PROGRAM P_SqlSelect
VAR
	
	fbSq : FB_EasySql;
	sSql : STRING(1000);
	
	iGE : INT:=1; //Select value
	
	astData : ARRAY[0..9] OF ST_SelectStruct; //Data array for recieved data
	
	bRead : BOOL; //Execute command
	bDone : BOOL; //Command done
	bError : BOOL; //Command error
	sError : STRING(255);
	
	udiNoOfRecords : UDINT; //Numbers of returned recoreds
	
END_VAR

//Select data from database
sSql := 'SELECT id,username,password FROM tpr_db.user where id >=¤1¤';

F_Replace(pString:= ADR(sSql), cbStringLen:= SIZEOF(sSql), sSearch:= '¤1¤', sReplace:= TO_STRING(iGE)); //Replace placeholder

fbSq(
	bExecute:= bRead, 
	wDBID:= 1, 
	pSql:= ADR(sSql), 
	cbSql:= SIZEOF(sSql), 
	pData:= ADR(astData), 
	cbData:= SIZEOF(astData), 
	udiMaxOfRecord:= 3, //Max number of recieved records
	udiNoOfRecords=> udiNoOfRecords, 
	bDone=> bDone, 
	bBusy=> , 
	bError=> bError, 
	sError=> sError
);

END_PROGRAM

(* stored: Version 1.1.0.1, ProductVersion 3.1.4024.4
   POU P_SqlSelect: Id {0c8a08bb-40b8-485a-9b2a-76a4d6dacfc7}, SpecialFunc None *)
